{attribute 'TcGenerated'}
{attribute 'no-analysis'}
{attribute 'linkalways'}
// This function has been automatically generated from the project information.
VAR_GLOBAL CONSTANT
	{attribute 'const_non_replaced'}
	stLibVersion_Tc3_CRC : ST_LibVersion := (iMajor := 0, iMinor := 0, iBuild := 0, iRevision := 1, nFlags := 0, sVersion := '0.0.0.1');
END_VAR

(* stored: Version 1.1.0.1
   GVL Global_Version: Id {e27c6247-4e28-411c-956a-46ad3aeabee5} *)
